// TIA Portal project "conveyor_automation" (V17)
// Vorlageprojekt für das Buch mit Zielsystem S7-1200

(* hardware
DEVICE "S7-1200-Station_1"  S7-1200 Station
   slot 0: "Baugruppenträger_0"  Rack  V1.0
   slot 1: "PLC_1"  CPU 1211C DC/DC/DC  6ES7 211-1AE40-0XB0  V4.1
*)

// ===== PLC "PLC_1"  CPU 1211C DC/DC/DC =====

VAR_GLOBAL   // PLC tag table "Standard-Variablentabelle"
   "Tag_1" AT %A0.0 : Bool;
   "Tag_2" AT %E0.0 : Bool;
   "Tag_3" AT %E0.1 : Bool;
   "conveyor_1" AT %Q0.2 : Bool;
   "conveyor_2" AT %Q0.3 : Bool;
   "conveyor_3" AT %Q0.4 : Bool;
   "sensor_1" AT %I0.5 : Bool;
   "sensor_2" AT %I0.6 : Bool;
   "sensor_3" AT %I0.7 : Bool;
   "start" AT %I1.0 : Bool;
   "stop" AT %I1.1 : Bool;
   "sys_stop" AT %M0.0 : Bool;
   "conveyors" AT %M0.1 : Bool;
   "Tag_4" AT %M0.2 : Bool;
   "tof_et" AT %MD2 : Time;
   "load_cell_1" AT %M0.3 : Bool;
   "Tag_5" AT %I1.2 : Bool;
   "Tag_6" AT %I1.3 : Bool;
   "Tag_7" AT %M0.4 : Bool;
   "curr_con" AT %Q0.5 : Bool;
   "prev_sensor" AT %I1.4 : Bool;
   "curr_sensor" AT %I1.5 : Bool;
   "next_sensor" AT %I1.6 : Bool;
   "run" AT %I1.7 : Bool;
   "run(1)" AT %Q0.6 : Bool;
   "run(2)" AT %Q0.7 : Bool;
   "reset_1" AT %I2.0 : Bool;
   "reset_2" AT %I2.1 : Bool;
   "reset_3" AT %I2.2 : Bool;
END_VAR

DATA_BLOCK "scl_block_DB"   // DB1
{ S7_Optimized_Access := 'TRUE' }
VERSION : 0.1
// stored: InstanceOfName middle_conveyors
"middle_conveyors"
BEGIN
END_DATA_BLOCK

DATA_BLOCK "scl_block_DB_1"   // DB2
{ S7_Optimized_Access := 'TRUE' }
VERSION : 0.1
// stored: InstanceOfName middle_conveyors
"middle_conveyors"
BEGIN
END_DATA_BLOCK

DATA_BLOCK "scl_block_DB_2"   // DB3
{ S7_Optimized_Access := 'TRUE' }
VERSION : 0.1
// stored: InstanceOfName middle_conveyors
"middle_conveyors"
BEGIN
END_DATA_BLOCK

DATA_BLOCK "first_conveyor_DB"   // DB4
{ S7_Optimized_Access := 'TRUE' }
VERSION : 0.1
// stored: InstanceOfName first_conveyor
"first_conveyor"
BEGIN
END_DATA_BLOCK

DATA_BLOCK "last_conveyor_DB"   // DB5
{ S7_Optimized_Access := 'TRUE' }
VERSION : 0.1
// stored: InstanceOfName last_conveyor
"last_conveyor"
BEGIN
END_DATA_BLOCK

DATA_BLOCK "1st_conveyor"   // DB6
{ S7_Optimized_Access := 'TRUE' }
VERSION : 0.1
// stored: InstanceOfName con_aut
"con_aut"
BEGIN
END_DATA_BLOCK

DATA_BLOCK "2nd_conveyor"   // DB7
{ S7_Optimized_Access := 'TRUE' }
VERSION : 0.1
// stored: InstanceOfName con_aut
"con_aut"
BEGIN
END_DATA_BLOCK

DATA_BLOCK "3rd_conveyor"   // DB8
{ S7_Optimized_Access := 'TRUE' }
VERSION : 0.1
// stored: InstanceOfName con_aut
"con_aut"
BEGIN
END_DATA_BLOCK

FUNCTION_BLOCK "first_conveyor"   // FB1, SCL
{ S7_Optimized_Access := 'TRUE' }
VERSION : 0.1
   VAR_INPUT
      curr_sensor : Bool;
      next_sensor : Bool;
   END_VAR
   VAR_OUTPUT
      curr_conveyor : Bool;
   END_VAR
BEGIN
   IF #curr_sensor = 1 AND #next_sensor = 0 THEN
       #curr_conveyor := 1;
   ELSIF #next_sensor = 1 AND #curr_sensor = 0 THEN
       #curr_conveyor := 0;
   ELSIF #curr_sensor = 1 AND #next_sensor = 1 THEN
       #curr_conveyor := 0;
   END_IF;
END_FUNCTION_BLOCK

FUNCTION_BLOCK "middle_conveyors"   // FB2, SCL
{ S7_Optimized_Access := 'TRUE' }
VERSION : 0.1
   VAR_INPUT
      next_sensor : Bool;
      curr_sensor : Bool;
      prev_sensor : Bool;
   END_VAR
   VAR_OUTPUT
      curr_conveyor : Bool;
   END_VAR
BEGIN
   IF #prev_sensor = 1 AND #curr_sensor = 0 THEN
       #curr_conveyor := 1;
   ELSIF #curr_sensor = 1 AND #next_sensor = 0 THEN
       #curr_conveyor := 1;
   ELSIF #prev_sensor = 1 AND #curr_sensor = 0 AND #next_sensor = 1 THEN
       #curr_conveyor := 1;
   ELSIF (#curr_sensor = 1 AND #next_sensor = 1) OR (#prev_sensor=0 AND #curr_sensor=0 AND #next_sensor=1) THEN
       #curr_conveyor := 0;
   END_IF;
END_FUNCTION_BLOCK

FUNCTION_BLOCK "last_conveyor"   // FB3, SCL
{ S7_Optimized_Access := 'TRUE' }
VERSION : 0.1
   VAR_INPUT
      prev_sensor : Bool;
      curr_sensor : Bool;
   END_VAR
   VAR_OUTPUT
      curr_conveyor : Bool;
   END_VAR
BEGIN
   IF #prev_sensor = 1 AND #curr_sensor = 0 THEN
       #curr_conveyor := 1;
   ELSIF #curr_sensor = 1 THEN
       #curr_conveyor := 0;
   END_IF;
END_FUNCTION_BLOCK

FUNCTION_BLOCK "con_aut"   // FB4, LAD
{ S7_Optimized_Access := 'TRUE' }
VERSION : 0.1
   VAR_INPUT
      prev_sensor : Bool;
      curr_sensor : Bool;
      next_sensor : Bool;
      reset : Bool;
   END_VAR
   VAR_OUTPUT
      curr_conveyor : Bool;
   END_VAR
   VAR
      run_stat : Bool;
      run_stat_2 : Bool;
      run_stat_3 : Bool;
      reset_stat : Bool;
   END_VAR
BEGIN

REGION Network 1
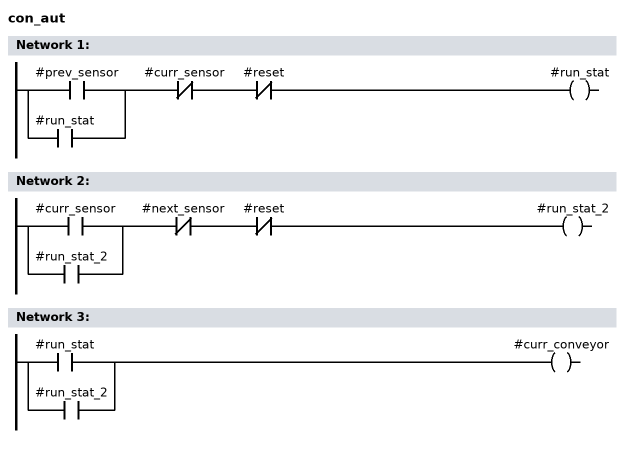
   RUNG wire#powerrail
      Contact( #prev_sensor )
      wire#w1
      I_Contact( #curr_sensor )
      I_Contact( #reset )
      Coil( #run_stat )
   END_RUNG
   RUNG wire#powerrail
      Contact( #run_stat )
   END_RUNG wire#w1
   // the same network as SCL:
   #run_stat := (#prev_sensor OR #run_stat) AND NOT #curr_sensor AND NOT #reset;
END_REGION

REGION Network 2
   RUNG wire#powerrail
      Contact( #curr_sensor )
      wire#w1
      I_Contact( #next_sensor )
      I_Contact( #reset )
      Coil( #run_stat_2 )
   END_RUNG
   RUNG wire#powerrail
      Contact( #run_stat_2 )
   END_RUNG wire#w1
   // the same network as SCL:
   #run_stat_2 := (#curr_sensor OR #run_stat_2) AND NOT #next_sensor AND NOT #reset;
END_REGION

REGION Network 3
   RUNG wire#powerrail
      Contact( #run_stat )
      wire#w1
      Coil( #curr_conveyor )
   END_RUNG
   RUNG wire#powerrail
      Contact( #run_stat_2 )
   END_RUNG wire#w1
   // the same network as SCL:
   #curr_conveyor := #run_stat OR #run_stat_2;
END_REGION
END_FUNCTION_BLOCK

FUNCTION "MHJ-PLC-Lab-Function-S71200" : Void   // FC9000, SCL
{ S7_Optimized_Access := 'TRUE' }
VERSION : 0.1
   VAR_TEMP
      rdTimeReturn : Int;
      outputTime : DTL;
      SyncVal : Byte;
      forVal : Int;
      forVal_2 : Int;
      Value : Byte;
   END_VAR
   VAR CONSTANT
      CompVal : Byte := 16#34;
      Value_01 : Byte := 16#11;
      Value_01_DW : DWord := 16#A165_D992;
      Value_02_DW : DWord := 16#58BE_4401;
   END_VAR
BEGIN

   #Value:=PEEK(area := 16#82,
        dbNumber := 0,
        byteOffset := 511);
   #Value := #Value + 1;

   POKE(area := 16#82,
        dbNumber := 0,
        byteOffset := 511,
        value := #Value);

   POKE(area:=16#81,
        dbNumber:=0,
        byteOffset:=1016,
        value:=#Value_01_DW);
   POKE(area := 16#81,
        dbNumber := 0,
        byteOffset := 1020,
        value := #Value_02_DW);

   POKE(area := 16#81,
        dbNumber := 0,
        byteOffset := 511,
        value := B#16#00);

   FOR #forVal := 0 TO 120 DO
       FOR #forVal_2:=0 TO 10 DO
           #rdTimeReturn:=RD_SYS_T(#outputTime);
           #rdTimeReturn := WR_SYS_T(#outputTime);
           #rdTimeReturn := RD_SYS_T(#outputTime);
           #rdTimeReturn := WR_SYS_T(#outputTime);
       END_FOR;
       #SyncVal:= PEEK(area := 16#81,
                      dbNumber := 0,
                      byteOffset := 511);
       IF #SyncVal = #CompVal THEN
          GOTO M_1;
       END_IF;
   END_FOR;
   RETURN;

   M_1:
   POKE(area := 16#81,
        dbNumber := 0,
        byteOffset := 511,
        value := B#16#0);
END_FUNCTION

ORGANIZATION_BLOCK "Main"   // OB1, LAD, ProgramCycle
TITLE = "Main Program Sweep (Cycle)"
{ S7_Optimized_Access := 'TRUE' }
VERSION : 0.1
   VAR_INPUT
      Initial_Call : Bool;   // Initial call of this OB
      Remanence : Bool;   // =True, if remanent data are available
   END_VAR
   VAR_TEMP   // added for the SCL form of the ladder/FBD networks
      _w1 : Bool;
   END_VAR
BEGIN

REGION Network 1: Konnektierungsbaustein für PLC-Lab
   // Im Netzwerk 1 wird der Konnektierungsbaustein für PLC-Lab aufgerufen.
   // Dieser Aufruf darf nicht entfernt werden!
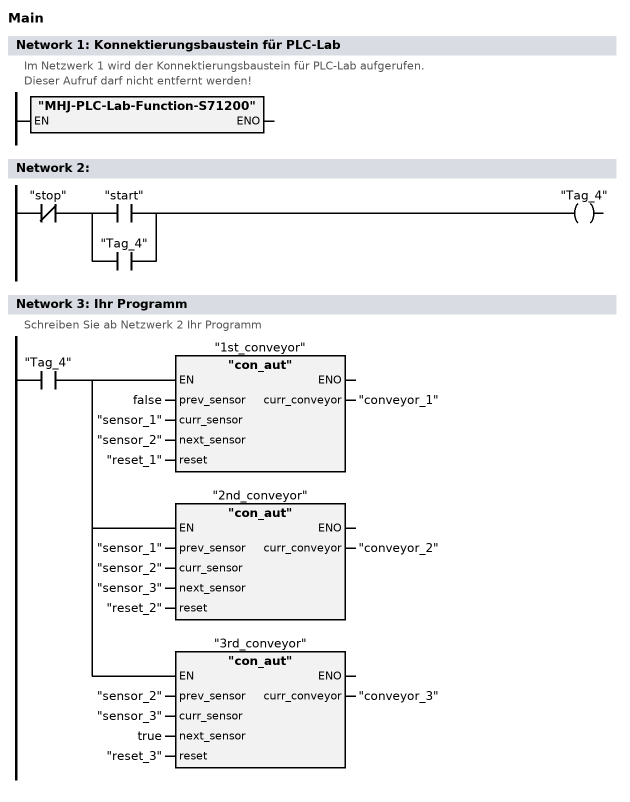
   RUNG wire#powerrail
      "MHJ-PLC-Lab-Function-S71200"()
   END_RUNG
   // the same network as SCL:
   "MHJ-PLC-Lab-Function-S71200"();
END_REGION

REGION Network 2
   RUNG wire#powerrail
      I_Contact( "stop" )
      wire#w1
      Contact( "start" )
      wire#w2
      Coil( "Tag_4" )
   END_RUNG
   RUNG wire#w1
      Contact( "Tag_4" )
   END_RUNG wire#w2
   // the same network as SCL:
   "Tag_4" := NOT "stop" AND ("start" OR "Tag_4");
END_REGION

REGION Network 3: Ihr Programm
   // Schreiben Sie ab Netzwerk 2 Ihr Programm
   RUNG wire#powerrail
      Contact( "Tag_4" )
      wire#w1
      "1st_conveyor"(prev_sensor := false, curr_sensor := "sensor_1", next_sensor := "sensor_2", reset := "reset_1", curr_conveyor => "conveyor_1")
   END_RUNG
   RUNG wire#w1
      "2nd_conveyor"(prev_sensor := "sensor_1", curr_sensor := "sensor_2", next_sensor := "sensor_3", reset := "reset_2", curr_conveyor => "conveyor_2")
   END_RUNG
   RUNG wire#w1
      "3rd_conveyor"(prev_sensor := "sensor_2", curr_sensor := "sensor_3", next_sensor := true, reset := "reset_3", curr_conveyor => "conveyor_3")
   END_RUNG
   // the same network as SCL:
   #_w1 := "Tag_4";
   IF #_w1 THEN
       "1st_conveyor"(prev_sensor := false,   // "con_aut"
                      curr_sensor := "sensor_1",
                      next_sensor := "sensor_2",
                      reset := "reset_1",
                      curr_conveyor => "conveyor_1");
       "2nd_conveyor"(prev_sensor := "sensor_1",   // "con_aut"
                      curr_sensor := "sensor_2",
                      next_sensor := "sensor_3",
                      reset := "reset_2",
                      curr_conveyor => "conveyor_2");
       "3rd_conveyor"(prev_sensor := "sensor_2",   // "con_aut"
                      curr_sensor := "sensor_3",
                      next_sensor := true,
                      reset := "reset_3",
                      curr_conveyor => "conveyor_3");
   END_IF;
END_REGION
END_ORGANIZATION_BLOCK